FUNCTION_BLOCK AUDI_AUI_MUX_32 (* AUDI multiplexor (generic FB) Adapter-Ausgang wird nur bei Wertänderung aktualisiert (Event nur bei tatsächlicher Änderung). *)
  (* Standard: 61499-2; Description: Copyright (c) 2026 HR Agrartechnik GmbH This program and the accompanying materials are made available under the terms of the Eclipse Public License 2.0 which is available at https://www.eclipse.org/legal/epl-2.0/ SPDX-License-Identifier: EPL-2.0 *)
  (* Version 1.0, 2026-08-13, Franz Höpfinger, HR Agrartechnik GmbH *)
  PACKAGE adapter::selection::unidirectional;
  {SET_ATTRIBUTE(eclipse4diac::core::GenericClassName, 'GEN_AUDI_AUI_MUX')}
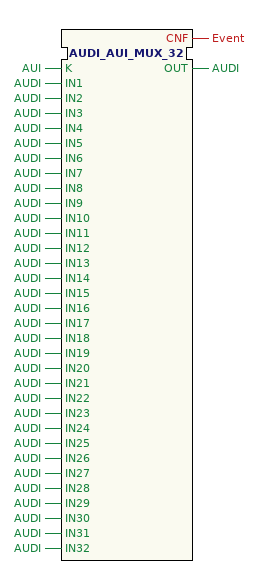
  EVENT_OUTPUT
    CNF; (* Confirmation of Set Index K *)
  END_EVENT
  SOCKETS
    K : adapter::types::unidirectional::AUI; (* index *)
    IN1 : adapter::types::unidirectional::AUDI; (* Input value 1 (selected when K = 0) *)
    IN2 : adapter::types::unidirectional::AUDI; (* Input value 2 (selected when K = 1) *)
    IN3 : adapter::types::unidirectional::AUDI; (* Input value 3 (selected when K = 2) *)
    IN4 : adapter::types::unidirectional::AUDI; (* Input value 4 (selected when K = 3) *)
    IN5 : adapter::types::unidirectional::AUDI; (* Input value 5 (selected when K = 4) *)
    IN6 : adapter::types::unidirectional::AUDI; (* Input value 6 (selected when K = 5) *)
    IN7 : adapter::types::unidirectional::AUDI; (* Input value 7 (selected when K = 6) *)
    IN8 : adapter::types::unidirectional::AUDI; (* Input value 8 (selected when K = 7) *)
    IN9 : adapter::types::unidirectional::AUDI; (* Input value 9 (selected when K = 8) *)
    IN10 : adapter::types::unidirectional::AUDI; (* Input value 10 (selected when K = 9) *)
    IN11 : adapter::types::unidirectional::AUDI; (* Input value 11 (selected when K = 10) *)
    IN12 : adapter::types::unidirectional::AUDI; (* Input value 12 (selected when K = 11) *)
    IN13 : adapter::types::unidirectional::AUDI; (* Input value 13 (selected when K = 12) *)
    IN14 : adapter::types::unidirectional::AUDI; (* Input value 14 (selected when K = 13) *)
    IN15 : adapter::types::unidirectional::AUDI; (* Input value 15 (selected when K = 14) *)
    IN16 : adapter::types::unidirectional::AUDI; (* Input value 16 (selected when K = 15) *)
    IN17 : adapter::types::unidirectional::AUDI; (* Input value 17 (selected when K = 16) *)
    IN18 : adapter::types::unidirectional::AUDI; (* Input value 18 (selected when K = 17) *)
    IN19 : adapter::types::unidirectional::AUDI; (* Input value 19 (selected when K = 18) *)
    IN20 : adapter::types::unidirectional::AUDI; (* Input value 20 (selected when K = 19) *)
    IN21 : adapter::types::unidirectional::AUDI; (* Input value 21 (selected when K = 20) *)
    IN22 : adapter::types::unidirectional::AUDI; (* Input value 22 (selected when K = 21) *)
    IN23 : adapter::types::unidirectional::AUDI; (* Input value 23 (selected when K = 22) *)
    IN24 : adapter::types::unidirectional::AUDI; (* Input value 24 (selected when K = 23) *)
    IN25 : adapter::types::unidirectional::AUDI; (* Input value 25 (selected when K = 24) *)
    IN26 : adapter::types::unidirectional::AUDI; (* Input value 26 (selected when K = 25) *)
    IN27 : adapter::types::unidirectional::AUDI; (* Input value 27 (selected when K = 26) *)
    IN28 : adapter::types::unidirectional::AUDI; (* Input value 28 (selected when K = 27) *)
    IN29 : adapter::types::unidirectional::AUDI; (* Input value 29 (selected when K = 28) *)
    IN30 : adapter::types::unidirectional::AUDI; (* Input value 30 (selected when K = 29) *)
    IN31 : adapter::types::unidirectional::AUDI; (* Input value 31 (selected when K = 30) *)
    IN32 : adapter::types::unidirectional::AUDI; (* Input value 32 (selected when K = 31) *)
  END_SOCKETS
  PLUGS
    OUT : adapter::types::unidirectional::AUDI; (* IN1 for K = 0..IN32 for K = 31 *)
  END_PLUGS
END_FUNCTION_BLOCK
